// TIA Portal project "Modbuclient" (V15)

(* hardware
DEVICE "S7-1200 station_1"  S7-1200 Station
   slot 0: "Rack_0"  S7-1200 Rack  Rack  V1.0
   slot 1: "PLC_1"  CPU 1214C DC/DC/DC  6ES7 214-1AG40-0XB0  V4.0
*)

// ===== PLC "PLC_1"  CPU 1214C DC/DC/DC =====

VAR_GLOBAL   // PLC tag table "Default tag table"
   "Clock_Byte" AT %MB0 : Byte;
   "Clock_10Hz" AT %M0.0 : Bool;
   "Clock_5Hz" AT %M0.1 : Bool;
   "Clock_2.5Hz" AT %M0.2 : Bool;
   "Clock_2Hz" AT %M0.3 : Bool;
   "Clock_1.25Hz" AT %M0.4 : Bool;
   "Clock_1Hz" AT %M0.5 : Bool;
   "Clock_0.625Hz" AT %M0.6 : Bool;
   "Clock_0.5Hz" AT %M0.7 : Bool;
   "Tag_1" AT %Q0.0 : Bool;
END_VAR

TYPE "User_data_type_1"
   STRUCT
      temperatura : Word;
   END_STRUCT;
END_TYPE

DATA_BLOCK "Modbusdata"   // DB2
{ S7_Optimized_Access := 'FALSE' }
VERSION : 0.1
   VAR
      Temperatura : Word;
      HoldingReg : Array[0..10] of Word;
   END_VAR
BEGIN
END_DATA_BLOCK

DATA_BLOCK "ModbusConfig"   // DB3
{ S7_Optimized_Access := 'TRUE' }
VERSION : 0.1
   VAR
      TCPConfig : TCON_IP_v4;
      Desconexion : Bool;
      IDconexion : UInt := 1;
      status : Word;
      Error : Bool;
      bUSY : Bool;
      DONE : Bool;
   END_VAR
BEGIN
   TCPConfig.InterfaceId := 64;
   TCPConfig.ID := 16#1;
   TCPConfig.RemoteAddress.ADDR[1] := 16#C0;
   TCPConfig.RemoteAddress.ADDR[2] := 16#A8;
   TCPConfig.RemoteAddress.ADDR[4] := 16#64;
   TCPConfig.RemotePort := 502;
   TCPConfig.ActiveEstablished := 1;
END_DATA_BLOCK

ORGANIZATION_BLOCK "Main"   // OB1, LAD, ProgramCycle
TITLE = "Main Program Sweep (Cycle)"
{ S7_Optimized_Access := 'TRUE' }
VERSION : 0.1
   VAR_INPUT
      Initial_Call : Bool;   // Initial call of this OB
      Remanence : Bool;   // =True, if remanent data are available
   END_VAR
BEGIN

REGION Network 1
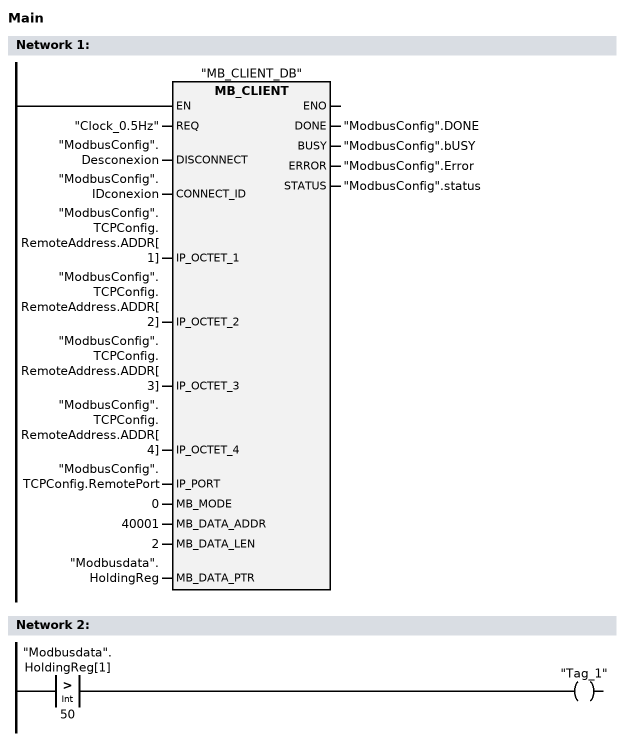
   "MB_CLIENT_DB"(REQ := "Clock_0.5Hz",   // MB_CLIENT
                  DISCONNECT := "ModbusConfig".Desconexion,
                  CONNECT_ID := "ModbusConfig".IDconexion,
                  IP_OCTET_1 := "ModbusConfig".TCPConfig.RemoteAddress.ADDR[1],
                  IP_OCTET_2 := "ModbusConfig".TCPConfig.RemoteAddress.ADDR[2],
                  IP_OCTET_3 := "ModbusConfig".TCPConfig.RemoteAddress.ADDR[3],
                  IP_OCTET_4 := "ModbusConfig".TCPConfig.RemoteAddress.ADDR[4],
                  IP_PORT := "ModbusConfig".TCPConfig.RemotePort,
                  MB_MODE := 0,
                  MB_DATA_ADDR := 40001,
                  MB_DATA_LEN := 2,
                  MB_DATA_PTR := "Modbusdata".HoldingReg,
                  DONE => "ModbusConfig".DONE,
                  BUSY => "ModbusConfig".bUSY,
                  ERROR => "ModbusConfig".Error,
                  STATUS => "ModbusConfig".status);
END_REGION

REGION Network 2
   RUNG wire#powerrail
      { S7_Templates := "SrcType := Int" } GT_Contact(in1 := "Modbusdata".HoldingReg[1], in2 := 50)
      Coil( "Tag_1" )
   END_RUNG
   // the same network as SCL:
   "Tag_1" := "Modbusdata".HoldingReg[1] > 50;
END_REGION
END_ORGANIZATION_BLOCK